       // === DIGITAL INPUTS: real %I bits -> IO_Buffer_DB.DI[1..368] ===
       // -- AFT DI modules --
       "IO_Buffer_DB".DI[1] := "Tag__639217692550262421";
       "IO_Buffer_DB".DI[2] := "Tag__639217692553776870";
       "IO_Buffer_DB".DI[3] := "Tag__639217692553954872";
       "IO_Buffer_DB".DI[4] := "Tag__639217692553954873";
       "IO_Buffer_DB".DI[5] := "Tag__639217692554216438";
       "IO_Buffer_DB".DI[6] := "Tag__639217692554394622";
       "IO_Buffer_DB".DI[7] := "Tag__639217692554432300";
       "IO_Buffer_DB".DI[8] := "Tag__639217692556336031";
       "IO_Buffer_DB".DI[9] := "Tag__639217692556550149";
       "IO_Buffer_DB".DI[10] := "Tag__639217692556680608";
       "IO_Buffer_DB".DI[11] := "Tag__639217692556821735";
       "IO_Buffer_DB".DI[12] := "Tag__639217692556891742";
       "IO_Buffer_DB".DI[13] := "Tag__639217692557049682";
       "IO_Buffer_DB".DI[14] := "Tag__639217692557209508";
       "IO_Buffer_DB".DI[15] := "Tag__639217692557209509";
       "IO_Buffer_DB".DI[16] := "Tag__639217692557471753";
       "IO_Buffer_DB".DI[17] := "Tag__639217692557529414";
       "IO_Buffer_DB".DI[18] := "Tag__639217692557689863";
       "IO_Buffer_DB".DI[19] := "Tag__639217692557850060";
       "IO_Buffer_DB".DI[20] := "Tag__639217692558010331";
       "IO_Buffer_DB".DI[21] := "Tag__639217692558171799";
       "IO_Buffer_DB".DI[22] := "Tag__639217692558331401";
       "IO_Buffer_DB".DI[23] := "Tag__639217692558488410";
       "IO_Buffer_DB".DI[24] := "Tag__639217692558802162";
       "IO_Buffer_DB".DI[25] := "Tag__639217692558961456";
       "IO_Buffer_DB".DI[26] := "Tag__639217692558971616";
       "IO_Buffer_DB".DI[27] := "Tag__639217692559129482";
       "IO_Buffer_DB".DI[28] := "Tag__639217692559281543";
       "IO_Buffer_DB".DI[29] := "Tag__639217692559443162";
       "IO_Buffer_DB".DI[30] := "Tag__639217692559601745";
       "IO_Buffer_DB".DI[31] := "Tag__639217692559760896";
       "IO_Buffer_DB".DI[32] := "Tag__639217692559921432";
       "IO_Buffer_DB".DI[33] := "Tag__639217692559921433";
       "IO_Buffer_DB".DI[34] := "Tag__639217692560082018";
       "IO_Buffer_DB".DI[35] := "Tag__639217692560402934";
       "IO_Buffer_DB".DI[36] := "Tag__639217692560402935";
       "IO_Buffer_DB".DI[37] := "Tag__639217692560583987";
       "IO_Buffer_DB".DI[38] := "Tag__639217692560723706";
       "IO_Buffer_DB".DI[39] := "Tag__639217692560880740";
       "IO_Buffer_DB".DI[40] := "Tag__639217692561041807";
       "IO_Buffer_DB".DI[41] := "Tag__639217692561206457";
       "IO_Buffer_DB".DI[42] := "Tag__639217692561359218";
       "IO_Buffer_DB".DI[43] := "Tag__639217692561520184";
       "IO_Buffer_DB".DI[44] := "Tag__639217692561520185";
       "IO_Buffer_DB".DI[45] := "Tag__639217692561802187";
       "IO_Buffer_DB".DI[46] := "Tag__639217692561935087";
       "IO_Buffer_DB".DI[47] := "Tag__639217692562065024";
       "IO_Buffer_DB".DI[48] := "Tag__639217692562223286";
       "IO_Buffer_DB".DI[49] := "Tag__639217692562383723";
       "IO_Buffer_DB".DI[50] := "Tag__639217692562543936";
       "IO_Buffer_DB".DI[51] := "Tag__639217692562543937";
       "IO_Buffer_DB".DI[52] := "Tag__639217692562862407";
       "IO_Buffer_DB".DI[53] := "Tag__639217692562862408";
       "IO_Buffer_DB".DI[54] := "Tag__639217692563093001";
       "IO_Buffer_DB".DI[55] := "Tag__639217692563182212";
       "IO_Buffer_DB".DI[56] := "Tag__639217692563343596";
       "IO_Buffer_DB".DI[57] := "Tag__639217692563511187";
       "IO_Buffer_DB".DI[58] := "Tag__639217692563662093";
       "IO_Buffer_DB".DI[59] := "Tag__639217692563662094";
       "IO_Buffer_DB".DI[60] := "Tag__639217692563823907";
       "IO_Buffer_DB".DI[61] := "Tag__639217692566083593";
       "IO_Buffer_DB".DI[62] := "Tag__639217692566201557";
       "IO_Buffer_DB".DI[63] := "Tag__639217692566360040";
       "IO_Buffer_DB".DI[64] := "Tag__639217692566517145";
       "IO_Buffer_DB".DI[65] := "Tag__639217692566674032";
       "IO_Buffer_DB".DI[66] := "Tag__639217692566832496";
       "IO_Buffer_DB".DI[67] := "Tag__639217692566832497";
       "IO_Buffer_DB".DI[68] := "Tag__639217692567184922";
       "IO_Buffer_DB".DI[69] := "Tag__639217692567336780";
       "IO_Buffer_DB".DI[70] := "Tag__639217692567388945";
       "IO_Buffer_DB".DI[71] := "Tag__639217692567546587";
       "IO_Buffer_DB".DI[72] := "Tag__639217692567707146";
       "IO_Buffer_DB".DI[73] := "Tag__639217692567868007";
       "IO_Buffer_DB".DI[74] := "Tag__639217692567868008";
       "IO_Buffer_DB".DI[75] := "Tag__639217692568025035";
       "IO_Buffer_DB".DI[76] := "Tag__639217692568182907";
       "IO_Buffer_DB".DI[77] := "Tag__639217692568341074";
       "IO_Buffer_DB".DI[78] := "Tag__639217692568550097";
       "IO_Buffer_DB".DI[79] := "Tag__639217692568683019";
       "IO_Buffer_DB".DI[80] := "Tag__639217692568840948";
       "IO_Buffer_DB".DI[81] := "Tag__639217692568971320";
       "IO_Buffer_DB".DI[82] := "Tag__639217692569119475";
       "IO_Buffer_DB".DI[83] := "Tag__639217692569298523";
       "IO_Buffer_DB".DI[84] := "Tag__639217692569460008";
       "IO_Buffer_DB".DI[85] := "Tag__639217692569619373";
       "IO_Buffer_DB".DI[86] := "Tag__639217692569780777";
       "IO_Buffer_DB".DI[87] := "Tag__639217692569780778";
       "IO_Buffer_DB".DI[88] := "Tag__639217692569942097";
       "IO_Buffer_DB".DI[89] := "Tag__639217692570102018";
       "IO_Buffer_DB".DI[90] := "Tag__639217692570262026";
       "IO_Buffer_DB".DI[91] := "Tag__639217692570422186";
       "IO_Buffer_DB".DI[92] := "Tag__639217692570422187";
       "IO_Buffer_DB".DI[93] := "Tag__639217692570583489";
       "IO_Buffer_DB".DI[94] := "Tag__639217692570745102";
       "IO_Buffer_DB".DI[95] := "Tag__639217692570906074";
       "IO_Buffer_DB".DI[96] := "Tag__639217692570906075";
       "IO_Buffer_DB".DI[97] := "Tag__639217692571063660";
       "IO_Buffer_DB".DI[98] := "Tag__639217692571223097";
       "IO_Buffer_DB".DI[99] := "Tag__639217692571384739";
       "IO_Buffer_DB".DI[100] := "Tag__639217692571544096";
       "IO_Buffer_DB".DI[101] := "Tag__639217692571703825";
       "IO_Buffer_DB".DI[102] := "Tag__639217692571865026";
       "IO_Buffer_DB".DI[103] := "Tag__639217692572024808";
       "IO_Buffer_DB".DI[104] := "Tag__639217692572184903";
       "IO_Buffer_DB".DI[105] := "Tag__639217692572395679";
       "IO_Buffer_DB".DI[106] := "Tag__639217692572536054";
       "IO_Buffer_DB".DI[107] := "Tag__639217692572670856";
       "IO_Buffer_DB".DI[108] := "Tag__639217692572707880";
       "IO_Buffer_DB".DI[109] := "Tag__639217692572861963";
       "IO_Buffer_DB".DI[110] := "Tag__639217692573067363";
       "IO_Buffer_DB".DI[111] := "Tag__639217692573180541";
       "IO_Buffer_DB".DI[112] := "Tag__639217692573357884";
       // -- MID DI modules --
       "IO_Buffer_DB".DI[113] := "Tag__639217692573503474";
       "IO_Buffer_DB".DI[114] := "Tag__639217692573503475";
       "IO_Buffer_DB".DI[115] := "Tag__639217692573691090";
       "IO_Buffer_DB".DI[116] := "Tag__639217692573812370";
       "IO_Buffer_DB".DI[117] := "Tag__639217692573973083";
       "IO_Buffer_DB".DI[118] := "Tag__639217692574133186";
       "IO_Buffer_DB".DI[119] := "Tag__639217692574289638";
       "IO_Buffer_DB".DI[120] := "Tag__639217692574448526";
       "IO_Buffer_DB".DI[121] := "Tag__639217692574609334";
       "IO_Buffer_DB".DI[122] := "Tag__639217692574768434";
       "IO_Buffer_DB".DI[123] := "Tag__639217692574930294";
       "IO_Buffer_DB".DI[124] := "Tag__639217692575083184";
       "IO_Buffer_DB".DI[125] := "Tag__639217692575261129";
       "IO_Buffer_DB".DI[126] := "Tag__639217692575419042";
       "IO_Buffer_DB".DI[127] := "Tag__639217692575539382";
       "IO_Buffer_DB".DI[128] := "Tag__639217692575911602";
       "IO_Buffer_DB".DI[129] := "Tag__639217692576029509";
       "IO_Buffer_DB".DI[130] := "Tag__639217692576029510";
       "IO_Buffer_DB".DI[131] := "Tag__639217692576190207";
       "IO_Buffer_DB".DI[132] := "Tag__639217692576351259";
       "IO_Buffer_DB".DI[133] := "Tag__639217692576511022";
       "IO_Buffer_DB".DI[134] := "Tag__639217692576672087";
       "IO_Buffer_DB".DI[135] := "Tag__639217692576832345";
       "IO_Buffer_DB".DI[136] := "Tag__639217692576952866";
       "IO_Buffer_DB".DI[137] := "Tag__639217692576990475";
       "IO_Buffer_DB".DI[138] := "Tag__639217692577151896";
       "IO_Buffer_DB".DI[139] := "Tag__639217692577372028";
       "IO_Buffer_DB".DI[140] := "Tag__639217692577469814";
       "IO_Buffer_DB".DI[141] := "Tag__639217692577766896";
       "IO_Buffer_DB".DI[142] := "Tag__639217692577926746";
       "IO_Buffer_DB".DI[143] := "Tag__639217692578046402";
       "IO_Buffer_DB".DI[144] := "Tag__639217692578046403";
       "IO_Buffer_DB".DI[145] := "Tag__639217692578204423";
       "IO_Buffer_DB".DI[146] := "Tag__639217692578364346";
       "IO_Buffer_DB".DI[147] := "Tag__639217692578525327";
       "IO_Buffer_DB".DI[148] := "Tag__639217692578706091";
       "IO_Buffer_DB".DI[149] := "Tag__639217692578841403";
       "IO_Buffer_DB".DI[150] := "Tag__639217692579004858";
       "IO_Buffer_DB".DI[151] := "Tag__639217692579155731";
       "IO_Buffer_DB".DI[152] := "Tag__639217692579314254";
       "IO_Buffer_DB".DI[153] := "Tag__639217692579314255";
       "IO_Buffer_DB".DI[154] := "Tag__639217692579474584";
       "IO_Buffer_DB".DI[155] := "Tag__639217692579635203";
       "IO_Buffer_DB".DI[156] := "Tag__639217692579794995";
       "IO_Buffer_DB".DI[157] := "Tag__639217692579955090";
       "IO_Buffer_DB".DI[158] := "Tag__639217692580275677";
       "IO_Buffer_DB".DI[159] := "Tag__639217692580432274";
       "IO_Buffer_DB".DI[160] := "Tag__639217692580552766";
       "IO_Buffer_DB".DI[161] := "Tag__639217692580590363";
       "IO_Buffer_DB".DI[162] := "Tag__639217692580751532";
       "IO_Buffer_DB".DI[163] := "Tag__639217692580913166";
       "IO_Buffer_DB".DI[164] := "Tag__639217692581133835";
       "IO_Buffer_DB".DI[165] := "Tag__639217692581227406";
       "IO_Buffer_DB".DI[166] := "Tag__639217692581387294";
       "IO_Buffer_DB".DI[167] := "Tag__639217692581507780";
       "IO_Buffer_DB".DI[168] := "Tag__639217692581545371";
       "IO_Buffer_DB".DI[169] := "Tag__639217692581704532";
       "IO_Buffer_DB".DI[170] := "Tag__639217692581863905";
       "IO_Buffer_DB".DI[171] := "Tag__639217692581863906";
       "IO_Buffer_DB".DI[172] := "Tag__639217692582023588";
       "IO_Buffer_DB".DI[173] := "Tag__639217692582184822";
       "IO_Buffer_DB".DI[174] := "Tag__639217692582344335";
       "IO_Buffer_DB".DI[175] := "Tag__639217692582505209";
       "IO_Buffer_DB".DI[176] := "Tag__639217692582505210";
       "IO_Buffer_DB".DI[177] := "Tag__639217692582664098";
       "IO_Buffer_DB".DI[178] := "Tag__639217692582825326";
       "IO_Buffer_DB".DI[179] := "Tag__639217692582994863";
       "IO_Buffer_DB".DI[180] := "Tag__639217692583198482";
       "IO_Buffer_DB".DI[181] := "Tag__639217692583329182";
       "IO_Buffer_DB".DI[182] := "Tag__639217692583430354";
       "IO_Buffer_DB".DI[183] := "Tag__639217692583542618";
       "IO_Buffer_DB".DI[184] := "Tag__639217692583692939";
       "IO_Buffer_DB".DI[185] := "Tag__639217692585720764";
       "IO_Buffer_DB".DI[186] := "Tag__639217692585760931";
       "IO_Buffer_DB".DI[187] := "Tag__639217692585920591";
       "IO_Buffer_DB".DI[188] := "Tag__639217692586101165";
       "IO_Buffer_DB".DI[189] := "Tag__639217692586241395";
       "IO_Buffer_DB".DI[190] := "Tag__639217692586241396";
       "IO_Buffer_DB".DI[191] := "Tag__639217692586401865";
       "IO_Buffer_DB".DI[192] := "Tag__639217692586559348";
       "IO_Buffer_DB".DI[193] := "Tag__639217692586717642";
       "IO_Buffer_DB".DI[194] := "Tag__639217692586876705";
       "IO_Buffer_DB".DI[195] := "Tag__639217692587037050";
       "IO_Buffer_DB".DI[196] := "Tag__639217692587198156";
       "IO_Buffer_DB".DI[197] := "Tag__639217692587198157";
       "IO_Buffer_DB".DI[198] := "Tag__639217692587438593";
       "IO_Buffer_DB".DI[199] := "Tag__639217692587516326";
       "IO_Buffer_DB".DI[200] := "Tag__639217692587676973";
       "IO_Buffer_DB".DI[201] := "Tag__639217692587676974";
       "IO_Buffer_DB".DI[202] := "Tag__639217692587854158";
       "IO_Buffer_DB".DI[203] := "Tag__639217692587995295";
       "IO_Buffer_DB".DI[204] := "Tag__639217692588156000";
       "IO_Buffer_DB".DI[205] := "Tag__639217692588379878";
       "IO_Buffer_DB".DI[206] := "Tag__639217692588550268";
       "IO_Buffer_DB".DI[207] := "Tag__639217692588708101";
       "IO_Buffer_DB".DI[208] := "Tag__639217692588866833";
       "IO_Buffer_DB".DI[209] := "Tag__639217692589023179";
       "IO_Buffer_DB".DI[210] := "Tag__639217692589158483";
       "IO_Buffer_DB".DI[211] := "Tag__639217692589208458";
       "IO_Buffer_DB".DI[212] := "Tag__639217692589366891";
       "IO_Buffer_DB".DI[213] := "Tag__639217692589526977";
       "IO_Buffer_DB".DI[214] := "Tag__639217692589687241";
       "IO_Buffer_DB".DI[215] := "Tag__639217692589848658";
       "IO_Buffer_DB".DI[216] := "Tag__639217692589848659";
       "IO_Buffer_DB".DI[217] := "Tag__639217692590010039";
       "IO_Buffer_DB".DI[218] := "Tag__639217692590170658";
       "IO_Buffer_DB".DI[219] := "Tag__639217692590328833";
       "IO_Buffer_DB".DI[220] := "Tag__639217692590485955";
       "IO_Buffer_DB".DI[221] := "Tag__639217692590485956";
       "IO_Buffer_DB".DI[222] := "Tag__639217692590645258";
       "IO_Buffer_DB".DI[223] := "Tag__639217692590805752";
       "IO_Buffer_DB".DI[224] := "Tag__639217692590966425";
       // -- FWD DI modules --
       "IO_Buffer_DB".DI[225] := "Tag__639217692590966426";
       "IO_Buffer_DB".DI[226] := "Tag__639217692591127321";
       "IO_Buffer_DB".DI[227] := "Tag__639217692591285391";
       "IO_Buffer_DB".DI[228] := "Tag__639217692591446446";
       "IO_Buffer_DB".DI[229] := "Tag__639217692591605376";
       "IO_Buffer_DB".DI[230] := "Tag__639217692591923527";
       "IO_Buffer_DB".DI[231] := "Tag__639217692591923528";
       "IO_Buffer_DB".DI[232] := "Tag__639217692592084854";
       "IO_Buffer_DB".DI[233] := "Tag__639217692592246014";
       "IO_Buffer_DB".DI[234] := "Tag__639217692592406057";
       "IO_Buffer_DB".DI[235] := "Tag__639217692592406058";
       "IO_Buffer_DB".DI[236] := "Tag__639217692592567050";
       "IO_Buffer_DB".DI[237] := "Tag__639217692592727547";
       "IO_Buffer_DB".DI[238] := "Tag__639217692592888082";
       "IO_Buffer_DB".DI[239] := "Tag__639217692593114463";
       "IO_Buffer_DB".DI[240] := "Tag__639217692593206619";
       "IO_Buffer_DB".DI[241] := "Tag__639217692593364125";
       "IO_Buffer_DB".DI[242] := "Tag__639217692593535630";
       "IO_Buffer_DB".DI[243] := "Tag__639217692593656106";
       "IO_Buffer_DB".DI[244] := "Tag__639217692593702147";
       "IO_Buffer_DB".DI[245] := "Tag__639217692593935520";
       "IO_Buffer_DB".DI[246] := "Tag__639217692594074769";
       "IO_Buffer_DB".DI[247] := "Tag__639217692594204786";
       "IO_Buffer_DB".DI[248] := "Tag__639217692594204787";
       "IO_Buffer_DB".DI[249] := "Tag__639217692594365259";
       "IO_Buffer_DB".DI[250] := "Tag__639217692594522265";
       "IO_Buffer_DB".DI[251] := "Tag__639217692594681744";
       "IO_Buffer_DB".DI[252] := "Tag__639217692594681745";
       "IO_Buffer_DB".DI[253] := "Tag__639217692594842324";
       "IO_Buffer_DB".DI[254] := "Tag__639217692595003601";
       "IO_Buffer_DB".DI[255] := "Tag__639217692595162932";
       "IO_Buffer_DB".DI[256] := "Tag__639217692595295217";
       "IO_Buffer_DB".DI[257] := "Tag__639217692595321829";
       "IO_Buffer_DB".DI[258] := "Tag__639217692595479808";
       "IO_Buffer_DB".DI[259] := "Tag__639217692595637197";
       "IO_Buffer_DB".DI[260] := "Tag__639217692595797438";
       "IO_Buffer_DB".DI[261] := "Tag__639217692595959028";
       "IO_Buffer_DB".DI[262] := "Tag__639217692596136048";
       "IO_Buffer_DB".DI[263] := "Tag__639217692596337735";
       "IO_Buffer_DB".DI[264] := "Tag__639217692596435546";
       "IO_Buffer_DB".DI[265] := "Tag__639217692596435547";
       "IO_Buffer_DB".DI[266] := "Tag__639217692596596639";
       "IO_Buffer_DB".DI[267] := "Tag__639217692596754611";
       "IO_Buffer_DB".DI[268] := "Tag__639217692596914545";
       "IO_Buffer_DB".DI[269] := "Tag__639217692597075234";
       "IO_Buffer_DB".DI[270] := "Tag__639217692597075235";
       "IO_Buffer_DB".DI[271] := "Tag__639217692597235934";
       "IO_Buffer_DB".DI[272] := "Tag__639217692597397011";
       "IO_Buffer_DB".DI[273] := "Tag__639217692597554180";
       "IO_Buffer_DB".DI[274] := "Tag__639217692597711217";
       "IO_Buffer_DB".DI[275] := "Tag__639217692597871107";
       "IO_Buffer_DB".DI[276] := "Tag__639217692598028494";
       "IO_Buffer_DB".DI[277] := "Tag__639217692598185471";
       "IO_Buffer_DB".DI[278] := "Tag__639217692598185472";
       "IO_Buffer_DB".DI[279] := "Tag__639217692598345589";
       "IO_Buffer_DB".DI[280] := "Tag__639217692598572817";
       "IO_Buffer_DB".DI[281] := "Tag__639217692598703247";
       "IO_Buffer_DB".DI[282] := "Tag__639217692598865809";
       "IO_Buffer_DB".DI[283] := "Tag__639217692599003448";
       "IO_Buffer_DB".DI[284] := "Tag__639217692599080153";
       "IO_Buffer_DB".DI[285] := "Tag__639217692599295021";
       "IO_Buffer_DB".DI[286] := "Tag__639217692599434105";
       "IO_Buffer_DB".DI[287] := "Tag__639217692599574585";
       "IO_Buffer_DB".DI[288] := "Tag__639217692599692113";
       "IO_Buffer_DB".DI[289] := "Tag__639217692599852177";
       "IO_Buffer_DB".DI[290] := "Tag__639217692599852178";
       "IO_Buffer_DB".DI[291] := "Tag__639217692600013096";
       "IO_Buffer_DB".DI[292] := "Tag__639217692600225652";
       "IO_Buffer_DB".DI[293] := "Tag__639217692600329437";
       "IO_Buffer_DB".DI[294] := "Tag__639217692600517312";
       "IO_Buffer_DB".DI[295] := "Tag__639217692600648060";
       "IO_Buffer_DB".DI[296] := "Tag__639217692600809555";
       "IO_Buffer_DB".DI[297] := "Tag__639217692600970188";
       "IO_Buffer_DB".DI[298] := "Tag__639217692600970189";
       "IO_Buffer_DB".DI[299] := "Tag__639217692601290117";
       "IO_Buffer_DB".DI[300] := "Tag__639217692601576181";
       "IO_Buffer_DB".DI[301] := "Tag__639217692601764420";
       "IO_Buffer_DB".DI[302] := "Tag__639217692601904130";
       "IO_Buffer_DB".DI[303] := "Tag__639217692601921632";
       "IO_Buffer_DB".DI[304] := "Tag__639217692602082038";
       "IO_Buffer_DB".DI[305] := "Tag__639217692602243355";
       "IO_Buffer_DB".DI[306] := "Tag__639217692602403696";
       "IO_Buffer_DB".DI[307] := "Tag__639217692602403697";
       "IO_Buffer_DB".DI[308] := "Tag__639217692602561458";
       "IO_Buffer_DB".DI[309] := "Tag__639217692602720965";
       "IO_Buffer_DB".DI[310] := "Tag__639217692602881697";
       "IO_Buffer_DB".DI[311] := "Tag__639217692602881698";
       "IO_Buffer_DB".DI[312] := "Tag__639217692603041227";
       "IO_Buffer_DB".DI[313] := "Tag__639217692603201062";
       "IO_Buffer_DB".DI[314] := "Tag__639217692603432857";
       "IO_Buffer_DB".DI[315] := "Tag__639217692603526128";
       "IO_Buffer_DB".DI[316] := "Tag__639217692603677627";
       "IO_Buffer_DB".DI[317] := "Tag__639217692603839177";
       "IO_Buffer_DB".DI[318] := "Tag__639217692603998759";
       "IO_Buffer_DB".DI[319] := "Tag__639217692603998760";
       "IO_Buffer_DB".DI[320] := "Tag__639217692604301271";
       "IO_Buffer_DB".DI[321] := "Tag__639217692604446823";
       "IO_Buffer_DB".DI[322] := "Tag__639217692604524554";
       "IO_Buffer_DB".DI[323] := "Tag__639217692604674613";
       "IO_Buffer_DB".DI[324] := "Tag__639217692604834416";
       "IO_Buffer_DB".DI[325] := "Tag__639217692605944492";
       "IO_Buffer_DB".DI[326] := "Tag__639217692606105425";
       "IO_Buffer_DB".DI[327] := "Tag__639217692606105426";
       "IO_Buffer_DB".DI[328] := "Tag__639217692606285541";
       "IO_Buffer_DB".DI[329] := "Tag__639217692606426194";
       "IO_Buffer_DB".DI[330] := "Tag__639217692606584564";
       "IO_Buffer_DB".DI[331] := "Tag__639217692606742338";
       "IO_Buffer_DB".DI[332] := "Tag__639217692606904136";
       "IO_Buffer_DB".DI[333] := "Tag__639217692607062435";
       "IO_Buffer_DB".DI[334] := "Tag__639217692607224125";
       "IO_Buffer_DB".DI[335] := "Tag__639217692607224126";
       "IO_Buffer_DB".DI[336] := "Tag__639217692607485341";
       "IO_Buffer_DB".DI[337] := "Tag__639217692607543000";
       "IO_Buffer_DB".DI[338] := "Tag__639217692607763945";
       "IO_Buffer_DB".DI[339] := "Tag__639217692607861770";
       "IO_Buffer_DB".DI[340] := "Tag__639217692608018680";
       "IO_Buffer_DB".DI[341] := "Tag__639217692608018681";
       "IO_Buffer_DB".DI[342] := "Tag__639217692608238678";
       "IO_Buffer_DB".DI[343] := "Tag__639217692608335365";
       "IO_Buffer_DB".DI[344] := "Tag__639217692608493637";
       "IO_Buffer_DB".DI[345] := "Tag__639217692608653174";
       "IO_Buffer_DB".DI[346] := "Tag__639217692608812275";
       "IO_Buffer_DB".DI[347] := "Tag__639217692608812276";
       "IO_Buffer_DB".DI[348] := "Tag__639217692609128733";
       "IO_Buffer_DB".DI[349] := "Tag__639217692609128734";
       "IO_Buffer_DB".DI[350] := "Tag__639217692609289890";
       "IO_Buffer_DB".DI[351] := "Tag__639217692609532283";
       "IO_Buffer_DB".DI[352] := "Tag__639217692609702548";
       "IO_Buffer_DB".DI[353] := "Tag__639217692609862538";
       "IO_Buffer_DB".DI[354] := "Tag__639217692609862539";
       "IO_Buffer_DB".DI[355] := "Tag__639217692610182631";
       "IO_Buffer_DB".DI[356] := "Tag__639217692610182632";
       "IO_Buffer_DB".DI[357] := "Tag__639217692610403611";
       "IO_Buffer_DB".DI[358] := "Tag__639217692610501805";
       "IO_Buffer_DB".DI[359] := "Tag__639217692610661275";
       "IO_Buffer_DB".DI[360] := "Tag__639217692610661276";
       "IO_Buffer_DB".DI[361] := "Tag__639217692610983046";
       "IO_Buffer_DB".DI[362] := "Tag__639217692610983047";
       "IO_Buffer_DB".DI[363] := "Tag__639217692611192346";
       "IO_Buffer_DB".DI[364] := "Tag__639217692611310653";
       "IO_Buffer_DB".DI[365] := "Tag__639217692611461334";
       "IO_Buffer_DB".DI[366] := "Tag__639217692611622448";
       "IO_Buffer_DB".DI[367] := "Tag__639217692611781748";
       "IO_Buffer_DB".DI[368] := "Tag__639217692611781749";

       // === DIGITAL OUTPUTS: IO_Buffer_DB.DQ[1..208] -> real %Q bits ===
       // -- AFT DQ modules --
       "Tag__639217692612263475" := "IO_Buffer_DB".DQ[1];
       "Tag__639217692612423650" := "IO_Buffer_DB".DQ[2];
       "Tag__639217692612585355" := "IO_Buffer_DB".DQ[3];
       "Tag__639217692612746418" := "IO_Buffer_DB".DQ[4];
       "Tag__639217692612905975" := "IO_Buffer_DB".DQ[5];
       "Tag__639217692612905976" := "IO_Buffer_DB".DQ[6];
       "Tag__639217692613224334" := "IO_Buffer_DB".DQ[7];
       "Tag__639217692613431048" := "IO_Buffer_DB".DQ[8];
       "Tag__639217692613549459" := "IO_Buffer_DB".DQ[9];
       "Tag__639217692613549460" := "IO_Buffer_DB".DQ[10];
       "Tag__639217692613700358" := "IO_Buffer_DB".DQ[11];
       "Tag__639217692613860481" := "IO_Buffer_DB".DQ[12];
       "Tag__639217692614018559" := "IO_Buffer_DB".DQ[13];
       "Tag__639217692614298000" := "IO_Buffer_DB".DQ[14];
       "Tag__639217692614480374" := "IO_Buffer_DB".DQ[15];
       "Tag__639217692614684823" := "IO_Buffer_DB".DQ[16];
       "Tag__639217692614993876" := "IO_Buffer_DB".DQ[17];
       "Tag__639217692615192661" := "IO_Buffer_DB".DQ[18];
       "Tag__639217692615372374" := "IO_Buffer_DB".DQ[19];
       "Tag__639217692615821386" := "IO_Buffer_DB".DQ[20];
       "Tag__639217692615982422" := "IO_Buffer_DB".DQ[21];
       "Tag__639217692616141851" := "IO_Buffer_DB".DQ[22];
       "Tag__639217692616362637" := "IO_Buffer_DB".DQ[23];
       "Tag__639217692616460481" := "IO_Buffer_DB".DQ[24];
       "Tag__639217692616782087" := "IO_Buffer_DB".DQ[25];
       "Tag__639217692616782088" := "IO_Buffer_DB".DQ[26];
       "Tag__639217692616940617" := "IO_Buffer_DB".DQ[27];
       "Tag__639217692617097153" := "IO_Buffer_DB".DQ[28];
       "Tag__639217692617257965" := "IO_Buffer_DB".DQ[29];
       "Tag__639217692617425635" := "IO_Buffer_DB".DQ[30];
       "Tag__639217692617581306" := "IO_Buffer_DB".DQ[31];
       "Tag__639217692617739154" := "IO_Buffer_DB".DQ[32];
       "Tag__639217692617899719" := "IO_Buffer_DB".DQ[33];
       "Tag__639217692618058569" := "IO_Buffer_DB".DQ[34];
       "Tag__639217692618215933" := "IO_Buffer_DB".DQ[35];
       "Tag__639217692618373391" := "IO_Buffer_DB".DQ[36];
       "Tag__639217692618554770" := "IO_Buffer_DB".DQ[37];
       "Tag__639217692618760680" := "IO_Buffer_DB".DQ[38];
       "Tag__639217692618931105" := "IO_Buffer_DB".DQ[39];
       "Tag__639217692619091004" := "IO_Buffer_DB".DQ[40];
       "Tag__639217692619165425" := "IO_Buffer_DB".DQ[41];
       "Tag__639217692619325369" := "IO_Buffer_DB".DQ[42];
       "Tag__639217692619487118" := "IO_Buffer_DB".DQ[43];
       "Tag__639217692619487119" := "IO_Buffer_DB".DQ[44];
       "Tag__639217692619648292" := "IO_Buffer_DB".DQ[45];
       "Tag__639217692619808948" := "IO_Buffer_DB".DQ[46];
       "Tag__639217692620036810" := "IO_Buffer_DB".DQ[47];
       "Tag__639217692620197299" := "IO_Buffer_DB".DQ[48];
       "Tag__639217692620337293" := "IO_Buffer_DB".DQ[49];
       "Tag__639217692620357294" := "IO_Buffer_DB".DQ[50];
       "Tag__639217692620515379" := "IO_Buffer_DB".DQ[51];
       "Tag__639217692620675332" := "IO_Buffer_DB".DQ[52];
       "Tag__639217692620835634" := "IO_Buffer_DB".DQ[53];
       "Tag__639217692620992973" := "IO_Buffer_DB".DQ[54];
       "Tag__639217692621152065" := "IO_Buffer_DB".DQ[55];
       "Tag__639217692621309565" := "IO_Buffer_DB".DQ[56];
       "Tag__639217692621469714" := "IO_Buffer_DB".DQ[57];
       "Tag__639217692621469715" := "IO_Buffer_DB".DQ[58];
       "Tag__639217692621630499" := "IO_Buffer_DB".DQ[59];
       "Tag__639217692621906549" := "IO_Buffer_DB".DQ[60];
       "Tag__639217692621950360" := "IO_Buffer_DB".DQ[61];
       "Tag__639217692622111179" := "IO_Buffer_DB".DQ[62];
       "Tag__639217692622292619" := "IO_Buffer_DB".DQ[63];
       "Tag__639217692622426875" := "IO_Buffer_DB".DQ[64];
       // -- MID DQ modules --
       "Tag__639217692622426876" := "IO_Buffer_DB".DQ[65];
       "Tag__639217692622587394" := "IO_Buffer_DB".DQ[66];
       "Tag__639217692622746975" := "IO_Buffer_DB".DQ[67];
       "Tag__639217692622906735" := "IO_Buffer_DB".DQ[68];
       "Tag__639217692623064209" := "IO_Buffer_DB".DQ[69];
       "Tag__639217692623222595" := "IO_Buffer_DB".DQ[70];
       "Tag__639217692623222596" := "IO_Buffer_DB".DQ[71];
       "Tag__639217692623428677" := "IO_Buffer_DB".DQ[72];
       "Tag__639217692623552568" := "IO_Buffer_DB".DQ[73];
       "Tag__639217692623706024" := "IO_Buffer_DB".DQ[74];
       "Tag__639217692623866625" := "IO_Buffer_DB".DQ[75];
       "Tag__639217692624026402" := "IO_Buffer_DB".DQ[76];
       "Tag__639217692624188100" := "IO_Buffer_DB".DQ[77];
       "Tag__639217692624296413" := "IO_Buffer_DB".DQ[78];
       "Tag__639217692624349590" := "IO_Buffer_DB".DQ[79];
       "Tag__639217692624607979" := "IO_Buffer_DB".DQ[80];
       "Tag__639217692624665644" := "IO_Buffer_DB".DQ[81];
       "Tag__639217692624979691" := "IO_Buffer_DB".DQ[82];
       "Tag__639217692625112094" := "IO_Buffer_DB".DQ[83];
       "Tag__639217692625921588" := "IO_Buffer_DB".DQ[84];
       "Tag__639217692626087431" := "IO_Buffer_DB".DQ[85];
       "Tag__639217692626253351" := "IO_Buffer_DB".DQ[86];
       "Tag__639217692626352897" := "IO_Buffer_DB".DQ[87];
       "Tag__639217692626510009" := "IO_Buffer_DB".DQ[88];
       "Tag__639217692626671657" := "IO_Buffer_DB".DQ[89];
       "Tag__639217692626671658" := "IO_Buffer_DB".DQ[90];
       "Tag__639217692626833520" := "IO_Buffer_DB".DQ[91];
       "Tag__639217692626994806" := "IO_Buffer_DB".DQ[92];
       "Tag__639217692627254988" := "IO_Buffer_DB".DQ[93];
       "Tag__639217692627312671" := "IO_Buffer_DB".DQ[94];
       "Tag__639217692627473354" := "IO_Buffer_DB".DQ[95];
       "Tag__639217692627673115" := "IO_Buffer_DB".DQ[96];
       "Tag__639217692627811109" := "IO_Buffer_DB".DQ[97];
       "Tag__639217692627949093" := "IO_Buffer_DB".DQ[98];
       "Tag__639217692628089666" := "IO_Buffer_DB".DQ[99];
       "Tag__639217692628107166" := "IO_Buffer_DB".DQ[100];
       "Tag__639217692628336120" := "IO_Buffer_DB".DQ[101];
       "Tag__639217692628492917" := "IO_Buffer_DB".DQ[102];
       "Tag__639217692628623290" := "IO_Buffer_DB".DQ[103];
       "Tag__639217692628761042" := "IO_Buffer_DB".DQ[104];
       "Tag__639217692628899816" := "IO_Buffer_DB".DQ[105];
       "Tag__639217692628972569" := "IO_Buffer_DB".DQ[106];
       "Tag__639217692629072663" := "IO_Buffer_DB".DQ[107];
       "Tag__639217692629316047" := "IO_Buffer_DB".DQ[108];
       "Tag__639217692629373725" := "IO_Buffer_DB".DQ[109];
       "Tag__639217692629533777" := "IO_Buffer_DB".DQ[110];
       "Tag__639217692629693574" := "IO_Buffer_DB".DQ[111];
       "Tag__639217692629851555" := "IO_Buffer_DB".DQ[112];
       "Tag__639217692630008442" := "IO_Buffer_DB".DQ[113];
       "Tag__639217692630168713" := "IO_Buffer_DB".DQ[114];
       "Tag__639217692630329520" := "IO_Buffer_DB".DQ[115];
       "Tag__639217692630490637" := "IO_Buffer_DB".DQ[116];
       "Tag__639217692630661059" := "IO_Buffer_DB".DQ[117];
       "Tag__639217692630807879" := "IO_Buffer_DB".DQ[118];
       "Tag__639217692630939597" := "IO_Buffer_DB".DQ[119];
       "Tag__639217692631073684" := "IO_Buffer_DB".DQ[120];
       "Tag__639217692631183654" := "IO_Buffer_DB".DQ[121];
       "Tag__639217692631183655" := "IO_Buffer_DB".DQ[122];
       "Tag__639217692631342517" := "IO_Buffer_DB".DQ[123];
       "Tag__639217692631504108" := "IO_Buffer_DB".DQ[124];
       "Tag__639217692631664286" := "IO_Buffer_DB".DQ[125];
       "Tag__639217692631824426" := "IO_Buffer_DB".DQ[126];
       "Tag__639217692631981364" := "IO_Buffer_DB".DQ[127];
       "Tag__639217692631981365" := "IO_Buffer_DB".DQ[128];
       // -- FWD DQ modules --
       "Tag__639217692632142556" := "IO_Buffer_DB".DQ[129];
       "Tag__639217692632301255" := "IO_Buffer_DB".DQ[130];
       "Tag__639217692632461403" := "IO_Buffer_DB".DQ[131];
       "Tag__639217692632622376" := "IO_Buffer_DB".DQ[132];
       "Tag__639217692632622377" := "IO_Buffer_DB".DQ[133];
       "Tag__639217692632781836" := "IO_Buffer_DB".DQ[134];
       "Tag__639217692633119556" := "IO_Buffer_DB".DQ[135];
       "Tag__639217692633257667" := "IO_Buffer_DB".DQ[136];
       "Tag__639217692633257668" := "IO_Buffer_DB".DQ[137];
       "Tag__639217692633606974" := "IO_Buffer_DB".DQ[138];
       "Tag__639217692633797544" := "IO_Buffer_DB".DQ[139];
       "Tag__639217692633935297" := "IO_Buffer_DB".DQ[140];
       "Tag__639217692634052982" := "IO_Buffer_DB".DQ[141];
       "Tag__639217692634250953" := "IO_Buffer_DB".DQ[142];
       "Tag__639217692634367505" := "IO_Buffer_DB".DQ[143];
       "Tag__639217692634526933" := "IO_Buffer_DB".DQ[144];
       "Tag__639217692634686575" := "IO_Buffer_DB".DQ[145];
       "Tag__639217692634847392" := "IO_Buffer_DB".DQ[146];
       "Tag__639217692635084699" := "IO_Buffer_DB".DQ[147];
       "Tag__639217692635166263" := "IO_Buffer_DB".DQ[148];
       "Tag__639217692635324026" := "IO_Buffer_DB".DQ[149];
       "Tag__639217692635482506" := "IO_Buffer_DB".DQ[150];
       "Tag__639217692635482507" := "IO_Buffer_DB".DQ[151];
       "Tag__639217692635642498" := "IO_Buffer_DB".DQ[152];
       "Tag__639217692635802017" := "IO_Buffer_DB".DQ[153];
       "Tag__639217692636027800" := "IO_Buffer_DB".DQ[154];
       "Tag__639217692636167857" := "IO_Buffer_DB".DQ[155];
       "Tag__639217692636298889" := "IO_Buffer_DB".DQ[156];
       "Tag__639217692636348888" := "IO_Buffer_DB".DQ[157];
       "Tag__639217692636549597" := "IO_Buffer_DB".DQ[158];
       "Tag__639217692636666551" := "IO_Buffer_DB".DQ[159];
       "Tag__639217692636827995" := "IO_Buffer_DB".DQ[160];
       "Tag__639217692636988786" := "IO_Buffer_DB".DQ[161];
       "Tag__639217692636988787" := "IO_Buffer_DB".DQ[162];
       "Tag__639217692637150621" := "IO_Buffer_DB".DQ[163];
       "Tag__639217692637311136" := "IO_Buffer_DB".DQ[164];
       "Tag__639217692637471435" := "IO_Buffer_DB".DQ[165];
       "Tag__639217692637631790" := "IO_Buffer_DB".DQ[166];
       "Tag__639217692637789494" := "IO_Buffer_DB".DQ[167];
       "Tag__639217692637950184" := "IO_Buffer_DB".DQ[168];
       "Tag__639217692637950185" := "IO_Buffer_DB".DQ[169];
       "Tag__639217692638109462" := "IO_Buffer_DB".DQ[170];
       "Tag__639217692638276714" := "IO_Buffer_DB".DQ[171];
       "Tag__639217692638427229" := "IO_Buffer_DB".DQ[172];
       "Tag__639217692638586533" := "IO_Buffer_DB".DQ[173];
       "Tag__639217692638747466" := "IO_Buffer_DB".DQ[174];
       "Tag__639217692638904386" := "IO_Buffer_DB".DQ[175];
       "Tag__639217692639063833" := "IO_Buffer_DB".DQ[176];
       "Tag__639217692639078981" := "IO_Buffer_DB".DQ[177];
       "Tag__639217692639243768" := "IO_Buffer_DB".DQ[178];
       "Tag__639217692639383298" := "IO_Buffer_DB".DQ[179];
       "Tag__639217692639542163" := "IO_Buffer_DB".DQ[180];
       "Tag__639217692639701541" := "IO_Buffer_DB".DQ[181];
       "Tag__639217692639892825" := "IO_Buffer_DB".DQ[182];
       "Tag__639217692640016631" := "IO_Buffer_DB".DQ[183];
       "Tag__639217692640016632" := "IO_Buffer_DB".DQ[184];
       "Tag__639217692640175734" := "IO_Buffer_DB".DQ[185];
       "Tag__639217692640332797" := "IO_Buffer_DB".DQ[186];
       "Tag__639217692640492541" := "IO_Buffer_DB".DQ[187];
       "Tag__639217692640652754" := "IO_Buffer_DB".DQ[188];
       "Tag__639217692640652755" := "IO_Buffer_DB".DQ[189];
       "Tag__639217692640812694" := "IO_Buffer_DB".DQ[190];
       "Tag__639217692640972759" := "IO_Buffer_DB".DQ[191];
       "Tag__639217692641133541" := "IO_Buffer_DB".DQ[192];
       "Tag__639217692641370581" := "IO_Buffer_DB".DQ[193];
       "Tag__639217692641539941" := "IO_Buffer_DB".DQ[194];
       "Tag__639217692641669868" := "IO_Buffer_DB".DQ[195];
       "Tag__639217692641679864" := "IO_Buffer_DB".DQ[196];
       "Tag__639217692641838308" := "IO_Buffer_DB".DQ[197];
       "Tag__639217692641998720" := "IO_Buffer_DB".DQ[198];
       "Tag__639217692642156578" := "IO_Buffer_DB".DQ[199];
       "Tag__639217692642313321" := "IO_Buffer_DB".DQ[200];
       "Tag__639217692642472571" := "IO_Buffer_DB".DQ[201];
       "Tag__639217692642631876" := "IO_Buffer_DB".DQ[202];
       "Tag__639217692642631877" := "IO_Buffer_DB".DQ[203];
       "Tag__639217692642792640" := "IO_Buffer_DB".DQ[204];
       "Tag__639217692642950472" := "IO_Buffer_DB".DQ[205];
       "Tag__639217692643191744" := "IO_Buffer_DB".DQ[206];
       "Tag__639217692643266837" := "IO_Buffer_DB".DQ[207];
       "Tag__639217692643431479" := "IO_Buffer_DB".DQ[208];
END_FUNCTION
